FUNCTION_BLOCK FB_CartCtrlSlowDown EXTENDS FB_CartCtrlBase
VAR_INPUT
END_VAR
VAR_OUTPUT
END_VAR
VAR

	m_tarPosInc: Vec8d;
	m_trajVel : Vec8d;
	m_initVel : Vec8d;
	m_initPos : Vec8d;
	m_initDec : Vec8d;
	
	//slow down and stop time
	m_incSlowStopTime :LREAL;
	m_slowStopTime :LREAL :=0.5;
	
	// filter cut-off frequency for cart drive force 
	m_cmdJoystickLpfCutoffFreq : LREAL :=8;
	m_cartCtrlFreq :LREAL:=8000;
END_VAR

// override this function in each exact controller
METHOD PROTECTED calcCmdJntPos : BOOL
VAR_IN_OUT CONSTANT
	// slave cart joint data
	i_slaveCart :FB_SlaveCart;
END_VAR

VAR
	i:INT;
END_VAR
//In this method, 5 represents the pillar postion , 6 represents the beam rotation angle ,7 represents the beam stretch position ,8 represents the overhang angle
m_incSlowStopTime :=LIMIT(0, m_incSlowStopTime + g_cartCtrlCycleTime, 1);

FOR i := 1 TO 8 BY 1 DO
	m_trajVel[i] := m_initVel[i] - m_initDec[i] * m_incSlowStopTime;
	IF ABS(m_initVel[i]) < ABS(m_initDec[i]) * m_incSlowStopTime THEN
		m_trajVel[i]:=0;
	END_IF
	m_tarPosInc[i] := m_tarPosInc[i] + m_trajVel[i] * g_cartCtrlCycleTime;
	m_cmdJntPos[i] := m_initPos[i] + m_tarPosInc[i];
END_FOR

IF m_incSlowStopTime >= m_slowStopTime THEN//m_slowStopTime THEN
	m_isFinished := TRUE;
END_IF
END_METHOD

// override this function in each exact controller
// NOTICE: set joint control mode here, and do some initialization if needed
METHOD PUBLIC init : BOOL
VAR_IN_OUT CONSTANT
	i_slaveCart	:FB_SlaveCart;
END_VAR
VAR_IN_OUT 
	r_cartCtrlCmd :ST_SlaveArmCtrlCmds;
END_VAR

m_cmdJntPos:=r_cartCtrlCmd.m_cmdJntPos;
m_initPos := m_cmdJntPos;

m_jntEnableFlag :=r_cartCtrlCmd.m_jntEnableFlag;

m_jntOPMode[5]:= DriverOPMode_cspMZ;
m_jntOPMode[6]:= DriverOPMode_Pos;
m_jntOPMode[7]:= DriverOPMode_Pos;
m_jntOPMode[8]:= DriverOPMode_Pos;

m_trajVel[5] := 0;
m_trajVel[6] := 0;
m_trajVel[7] := 0;
m_trajVel[8] := 0;

m_tarPosInc[5] := 0;
m_tarPosInc[6] := 0;
m_tarPosInc[7] := 0;
m_tarPosInc[8] := 0;


m_incSlowStopTime := 0;

m_initVel[5] := LIMIT(-GVL_CartMotorParameters.g_maxJntVel[5], i_slaveCart.curJntVel[5], GVL_CartMotorParameters.g_maxJntVel[5]);
m_initVel[6] := LIMIT(-GVL_CartMotorParameters.g_maxJntVel[6], i_slaveCart.curJntVel[6], GVL_CartMotorParameters.g_maxJntVel[6]);
m_initVel[7] := LIMIT(-GVL_CartMotorParameters.g_maxJntVel[7], i_slaveCart.curJntVel[7], GVL_CartMotorParameters.g_maxJntVel[7]);
m_initVel[8] := LIMIT(-GVL_CartMotorParameters.g_maxJntVel[8], i_slaveCart.curJntVel[8], GVL_CartMotorParameters.g_maxJntVel[8]);


m_initDec[5] := sign(m_initVel[5])*GVL_CartMotorParameters.g_maxJntVel[5];
m_initDec[6] := sign(m_initVel[6])*GVL_CartMotorParameters.g_maxJntVel[6];
m_initDec[7] := sign(m_initVel[7])*GVL_CartMotorParameters.g_maxJntVel[7];
m_initDec[8] := sign(m_initVel[8])*GVL_CartMotorParameters.g_maxJntVel[8];


m_slowStopTime := 0.5;
// update commands to arm
copyCmds(r_cartCtrlCmd);
END_METHOD

END_FUNCTION_BLOCK

(* stored: Version 1.1.0.1, ProductVersion 3.1.4024.11
   POU FB_CartCtrlSlowDown: Id {0c77f5f0-20e1-4fb9-8be8-91bb56c7cc44}, SpecialFunc None
   Method calcCmdJntPos: Id {630fb5ab-8a03-4b8b-9301-f4144cd8fed1}
   Method init: Id {1889fc8b-7615-4a73-af47-9f6b2589ad8d} *)
